// Mitsubishi GX Works2 project: IELET2103_Datalab3   PLC: FX2N/FX2NC
// IELET2103_Datalab3

// global labels: Global1
VAR_GLOBAL
  StoppM1 : BOOL;
  StartM1 : BOOL;
  MotorvernM1 : BOOL;
  MotorM1 : BOOL;
  StoppM2 : BOOL;
  StartM2 : BOOL;
  MotorvernM2 : BOOL;
  MotorM2 : BOOL;
END_VAR

// task Task_01 (event TRUE, interval 0, priority 31): Oppgave3

PROGRAM Oppgave1b)
(* structured ladder/FBD written out as ST: instructions are called as NAME(EN, inputs, outputs); _pN, _eN, _tN stand for wires *)
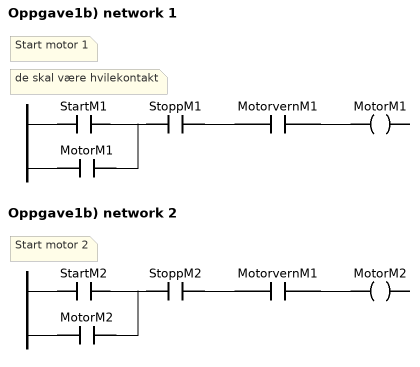
(* network 1 *)
(* Start motor 1 *)
(* de skal være hvilekontakt *)
MotorM1 := ((StartM1 OR MotorM1) AND StoppM1) AND MotorvernM1;
(* network 2 *)
(* Start motor 2 *)
MotorM2 := ((StartM2 OR MotorM2) AND StoppM2) AND MotorvernM1;
END_PROGRAM

FUNCTION_BLOCK Motorstart
VAR_INPUT
  Start : BOOL;
  Stopp : BOOL;
  Motorvern : BOOL;
END_VAR
VAR_OUTPUT
  Motor : BOOL;
END_VAR
(* structured ladder/FBD written out as ST: instructions are called as NAME(EN, inputs, outputs); _pN, _eN, _tN stand for wires *)
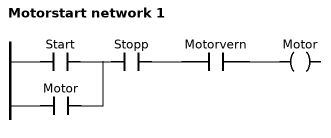
(* network 1 *)
Motor := ((Start OR Motor) AND Stopp) AND Motorvern;
END_FUNCTION_BLOCK

PROGRAM Oppgave2
VAR
  Motor_1 : Motorstart;
  Motor_2 : Motorstart;
END_VAR
(* structured ladder/FBD written out as ST: instructions are called as NAME(EN, inputs, outputs); _pN, _eN, _tN stand for wires *)
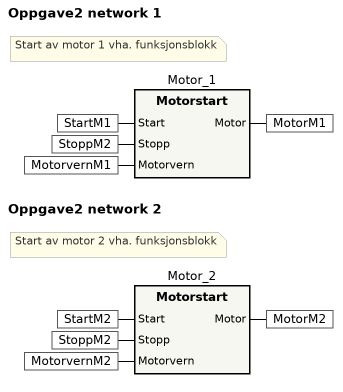
(* network 1 *)
(* Start av motor 1 vha. funksjonsblokk *)
Motor_1(Start := StartM1, Stopp := StoppM2, Motorvern := MotorvernM1, Motor => MotorM1);
(* network 2 *)
(* Start av motor 2 vha. funksjonsblokk *)
Motor_2(Start := StartM2, Stopp := StoppM2, Motorvern := MotorvernM2, Motor => MotorM2);
END_PROGRAM

PROGRAM Oppgave3
VAR
  Startflagg : BOOL;
  UforutsetteStopp : BOOL;
  Kvittert : BOOL;
END_VAR
(* structured ladder/FBD written out as ST: instructions are called as NAME(EN, inputs, outputs); _pN, _eN, _tN stand for wires *)
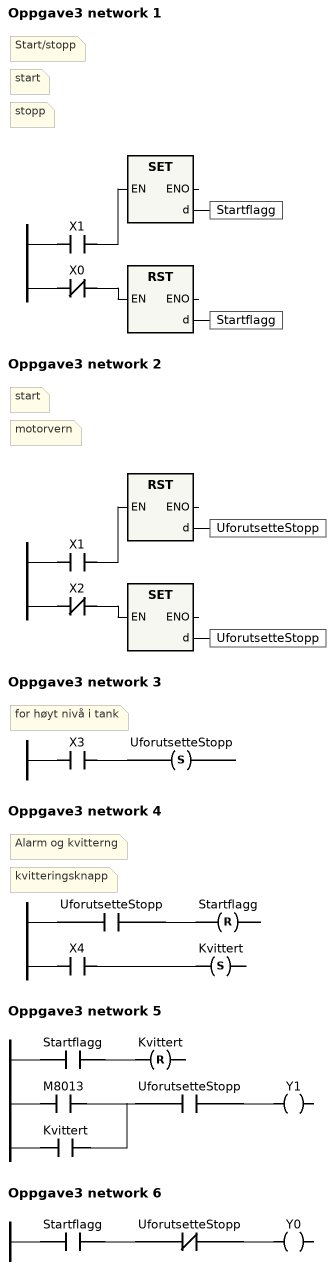
(* network 1 *)
(* Start/stopp *)
(* start *)
(* stopp *)
SET(X1, Startflagg);
RST(NOT X0, Startflagg);
(* network 2 *)
(* start *)
(* motorvern *)
RST(X1, UforutsetteStopp);
SET(NOT X2, UforutsetteStopp);
(* network 3 *)
(* for høyt nivå i tank *)
SET(X3, UforutsetteStopp);
(* network 4 *)
(* Alarm og kvitterng *)
(* kvitteringsknapp *)
RST(UforutsetteStopp, Startflagg);
SET(X4, Kvittert);
(* network 5 *)
RST(Startflagg, Kvittert);
Y1 := (M8013 OR Kvittert) AND UforutsetteStopp;
(* network 6 *)
Y0 := Startflagg AND NOT UforutsetteStopp;
END_PROGRAM
